TYPE "FCP_STATUS_WORD"
VERSION : 0.1
// Block: FCP_STATUS_WORD
   STRUCT
      Reserved0 : Bool;
      Reserved1 : Bool;
      DoublePumpVgMin : Bool;
      PresDropCompensation : Bool;
      PresCmdReached : Bool;
      Status : Bool;
      Warning : Bool;
      Error : Bool;
      Reserved8 : Bool;
      Reserved9 : Bool;
      Slave : Bool;
      ParGroup1 : Bool;
      Reserved12 : Bool;
      Reserved13 : Bool;
      Reserved14 : Bool;
      Reserved15 : Bool;
   END_STRUCT;

END_TYPE
